# EPICS autosave request: measCompApp/Db/measCompPulseGen_settings.req
$(P)$(R)Period
$(P)$(R)Width
$(P)$(R)Delay
$(P)$(R)Count
$(P)$(R)IdleState
